// TIA Portal V16 export
// export: Created 2022-11-17T15:49:45.9581143Z, ExportSetting WithDefaults, DisplayName Totally Integrated Automation Portal, DisplayVersion V16 Update 6, DisplayName TIA Portal Version Control Interface, DisplayVersion V16 Update 2, DisplayName TIA Portal Openness, DisplayVersion V16 Update 6, DisplayName SINAMICS Startdrive Advanced, DisplayVersion V16 Update 5, DisplayName SINAMICS Startdrive G130, G150, S120, S150, SINAMICS MV, S210, DisplayVersion V16 Update 5, DisplayName SINAMICS Startdrive G110M, G120, G120C, G120D, G120P, G115D, DisplayVersion V16 Update 5, DisplayName STEP 7 Professional, DisplayVersion V16 Update 6, DisplayName STEP 7 Safety, DisplayVersion V16, DisplayName WinCC Advanced, DisplayVersion V16 Update 6
DATA_BLOCK "DB247_Program3"   // DB247
{ S7_Optimized_Access := 'FALSE' }
AUTHOR : Robopac
VERSION : 0.0
// stored: AutoNumber false, IsOnlyStoredInLoadMemory false, IsWriteProtectedInAS false
   VAR RETAIN
      Program3 { S7_SetPoint := 'True'} : "DatiProgramma";
   END_VAR
BEGIN
   Program3.Wrapping := TRUE;
   Program3.TopLenght := 500;
   Program3.TopRelease := 0;
   Program3.TopDown := 0;
   Program3.Top := 4;
   Program3.PressurePTime := 0;
   Program3.LifterTime := 0;
   Program3.RevOverContrast := 1;
   Program3.RopeEndCycle := 16#01;
   Program3.Spare4 := 16#01;
   Program3.RopeTime := 1500;
   Program3.RevOverClamp := 1;
   Program3.FilmForceFinalRev := 20;
   Program3.FilmPrestretchFinalRev := 100;
   Program3.ArmSpeed := 90;
   Program3.CarriageDown4Top := 500;
   Program3.TopDownTime := 1500;
   Program3.LapsUnderTop := 0;
   Program3.Spare6 := 0;
   Program3.Spare7 := 0;
   Program3.Spare8 := 0;
   Program3.Spare9 := 0;
   Program3.Spare10 := 0;
   Program3.Spare11 := 0;
   Program3.Spare12 := 0;
   Program3.Overlap0_1 := 0;
   Program3.Height1 := 120;
   Program3.Landmark1 := FALSE;
   Program3.Lifter1 := FALSE;
   Program3.SpareBit1H1 := FALSE;
   Program3.Airblower1 := TRUE;
   Program3.NextStep1 := TRUE;
   Program3.PressureP1 := TRUE;
   Program3.SpareByte2H1 := 16#00;
   Program3.Revolution1 := 1;
   Program3.RopeUnit1_1 := 16#01;
   Program3.RopeUnit1_2 := 16#01;
   Program3.FilmForce1 := 5;
   Program3.FilmPrestretch1 := 200;
   Program3.Spare3H1 := 0;
   Program3.Spare49 := 0;
   Program3.Spare50 := 0;
   Program3.Spare51 := 0;
   Program3.Spare52 := 0;
   Program3.Spare53 := 0;
   Program3.Overlap1_2 := 0;
   Program3.Height2 := 60;
   Program3.Landmark2 := FALSE;
   Program3.Lifter2 := FALSE;
   Program3.SpareBit1H2 := FALSE;
   Program3.Airblower2 := TRUE;
   Program3.NextStep2 := TRUE;
   Program3.PressureP2 := TRUE;
   Program3.SpareByte2H2 := 16#00;
   Program3.Revolution2 := 3;
   Program3.RopeUnit2_1 := 16#01;
   Program3.RopeUnit2_2 := 16#01;
   Program3.FilmForce2 := 10;
   Program3.FilmPrestretch2 := 200;
   Program3.Spare3H2 := 0;
   Program3.Spare54 := 0;
   Program3.Spare55 := 0;
   Program3.Spare56 := 0;
   Program3.Spare57 := 0;
   Program3.Spare58 := 0;
   Program3.Overlap2_3 := 100;
   Program3.Height3 := 120;
   Program3.Landmark3 := FALSE;
   Program3.Lifter3 := FALSE;
   Program3.SpareBit1H3 := FALSE;
   Program3.Airblower3 := TRUE;
   Program3.NextStep3 := TRUE;
   Program3.PressureP3 := TRUE;
   Program3.SpareByte2H3 := 16#00;
   Program3.Revolution3 := 2;
   Program3.RopeUnit3_1 := 16#01;
   Program3.RopeUnit3_2 := 16#01;
   Program3.FilmForce3 := 5;
   Program3.FilmPrestretch3 := 200;
   Program3.Spare3H3 := 0;
   Program3.Spare59 := 0;
   Program3.Spare60 := 0;
   Program3.Spare61 := 380;
   Program3.Spare62 := 2800;
   Program3.Spare63 := 0;
   Program3.Overlap3_4 := 200;
   Program3.Height4 := 120;
   Program3.Landmark4 := FALSE;
   Program3.Lifter4 := FALSE;
   Program3.SpareBit1H4 := FALSE;
   Program3.Airblower4 := TRUE;
   Program3.NextStep4 := TRUE;
   Program3.PressureP4 := TRUE;
   Program3.SpareByte2H4 := 16#00;
   Program3.Revolution4 := 1;
   Program3.RopeUnit4_1 := 16#01;
   Program3.RopeUnit4_2 := 16#01;
   Program3.FilmForce4 := 20;
   Program3.FilmPrestretch4 := 200;
   Program3.Spare3H4 := 0;
   Program3.Spare64 := 0;
   Program3.Spare65 := 0;
   Program3.Spare66 := 0;
   Program3.Spare67 := 0;
   Program3.Spare68 := 0;
   Program3.Overlap4_5 := 200;
   Program3.Height5 := -150;
   Program3.Landmark5 := TRUE;
   Program3.Lifter5 := FALSE;
   Program3.SpareBit1H5 := FALSE;
   Program3.Airblower5 := FALSE;
   Program3.NextStep5 := TRUE;
   Program3.PressureP5 := FALSE;
   Program3.SpareByte2H5 := 16#00;
   Program3.Revolution5 := 1;
   Program3.RopeUnit5_1 := 16#01;
   Program3.RopeUnit5_2 := 16#01;
   Program3.FilmForce5 := 20;
   Program3.FilmPrestretch5 := 200;
   Program3.Spare3H5 := 0;
   Program3.Spare69 := 0;
   Program3.Spare70 := 0;
   Program3.Spare71 := 0;
   Program3.Spare72 := 0;
   Program3.Spare73 := 0;
   Program3.Overlap5_6 := 100;
   Program3.Height6 := 0;
   Program3.Landmark6 := FALSE;
   Program3.Lifter6 := FALSE;
   Program3.SpareBit1H6 := FALSE;
   Program3.Airblower6 := FALSE;
   Program3.NextStep6 := FALSE;
   Program3.PressureP6 := FALSE;
   Program3.SpareByte2H6 := 16#00;
   Program3.Revolution6 := 1;
   Program3.RopeUnit6_1 := 16#01;
   Program3.RopeUnit6_2 := 16#01;
   Program3.FilmForce6 := 30;
   Program3.FilmPrestretch6 := 200;
   Program3.Spare3H6 := 0;
   Program3.Spare74 := 0;
   Program3.Spare75 := 0;
   Program3.Spare76 := 0;
   Program3.Spare77 := 0;
   Program3.Spare78 := 0;
   Program3.Overlap6_7 := 0;
   Program3.Height7 := 0;
   Program3.Landmark7 := FALSE;
   Program3.Lifter7 := FALSE;
   Program3.SpareBit1H7 := FALSE;
   Program3.Airblower7 := FALSE;
   Program3.NextStep7 := TRUE;
   Program3.PressureP7 := FALSE;
   Program3.SpareByte2H7 := 16#00;
   Program3.Revolution7 := 1;
   Program3.RopeUnit7_1 := 16#01;
   Program3.RopeUnit7_2 := 16#01;
   Program3.FilmForce7 := 0;
   Program3.FilmPrestretch7 := 100;
   Program3.Spare3H7 := 0;
   Program3.Spare79 := 0;
   Program3.Spare80 := 0;
   Program3.Spare81 := 0;
   Program3.Spare82 := 0;
   Program3.Spare83 := 0;
   Program3.Overlap7_8 := 0;
   Program3.Height8 := 0;
   Program3.Landmark8 := FALSE;
   Program3.Lifter8 := FALSE;
   Program3.SpareBit1H8 := FALSE;
   Program3.Airblower8 := FALSE;
   Program3.NextStep8 := TRUE;
   Program3.PressureP8 := FALSE;
   Program3.SpareByte2H8 := 16#00;
   Program3.Revolution8 := 1;
   Program3.RopeUnit8_1 := 16#01;
   Program3.RopeUnit8_2 := 16#01;
   Program3.FilmForce8 := 0;
   Program3.FilmPrestretch8 := 100;
   Program3.Spare3H8 := 0;
   Program3.Spare84 := 0;
   Program3.Spare85 := 0;
   Program3.Spare86 := 0;
   Program3.Spare87 := 0;
   Program3.Spare88 := 0;
   Program3.Overlap8_9 := 0;
   Program3.Height9 := 0;
   Program3.Landmark9 := FALSE;
   Program3.Lifter9 := FALSE;
   Program3.SpareBit1H9 := FALSE;
   Program3.Airblower9 := FALSE;
   Program3.NextStep9 := TRUE;
   Program3.PressureP9 := FALSE;
   Program3.SpareByte2H9 := 16#00;
   Program3.Revolution9 := 1;
   Program3.RopeUnit9_1 := 16#01;
   Program3.RopeUnit9_2 := 16#01;
   Program3.FilmForce9 := 0;
   Program3.FilmPrestretch9 := 100;
   Program3.Spare3H9 := 0;
   Program3.Spare89 := 0;
   Program3.Spare90 := 0;
   Program3.Spare91 := 0;
   Program3.Spare92 := 0;
   Program3.Spare93 := 0;
   Program3.Overlap9_10 := 0;
   Program3.Height10 := 0;
   Program3.Landmark10 := FALSE;
   Program3.Lifter10 := FALSE;
   Program3.SpareBit1H10 := FALSE;
   Program3.Airblower10 := FALSE;
   Program3.NextStep10 := FALSE;
   Program3.PressureP10 := FALSE;
   Program3.SpareByte2H10 := 16#00;
   Program3.Revolution10 := 1;
   Program3.RopeUnit10_1 := 16#01;
   Program3.RopeUnit10_2 := 16#01;
   Program3.FilmForce10 := 0;
   Program3.FilmPrestretch10 := 100;
   Program3.Spare3H10 := 0;
   Program3.Spare94 := 0;
   Program3.Spare95 := 0;
   Program3.Spare96 := 0;
   Program3.Spare97 := 0;
   Program3.Spare98 := 0;
   Program3.Overlap10_11 := 0;
   Program3.Height11 := 0;
   Program3.Landmark11 := FALSE;
   Program3.Lifter11 := FALSE;
   Program3.SpareBit1H11 := FALSE;
   Program3.Airblower11 := FALSE;
   Program3.NextStep11 := TRUE;
   Program3.PressureP11 := FALSE;
   Program3.SpareByte2H11 := 16#00;
   Program3.Revolution11 := 1;
   Program3.RopeUnit11_1 := 16#01;
   Program3.RopeUnit11_2 := 16#01;
   Program3.FilmForce11 := 0;
   Program3.FilmPrestretch11 := 100;
   Program3.Spare3H11 := 0;
   Program3.Spare99 := 0;
   Program3.Spare100 := 0;
   Program3.Spare101 := 0;
   Program3.Spare102 := 0;
   Program3.Spare103 := 0;
   Program3.Overlap11_12 := 0;
   Program3.Height12 := 0;
   Program3.Landmark12 := FALSE;
   Program3.Lifter12 := FALSE;
   Program3.SpareBit1H12 := FALSE;
   Program3.Airblower12 := FALSE;
   Program3.NextStep12 := FALSE;
   Program3.PressureP12 := FALSE;
   Program3.SpareByte2H12 := 16#00;
   Program3.Revolution12 := 1;
   Program3.RopeUnit12_1 := 16#01;
   Program3.RopeUnit12_2 := 16#01;
   Program3.FilmForce12 := 0;
   Program3.FilmPrestretch12 := 100;
   Program3.Spare3H12 := 0;
   Program3.Spare104 := 0;
   Program3.Spare105 := 0;
   Program3.Spare106 := 0;
   Program3.Spare107 := 0;
   Program3.Spare108 := 0;
END_DATA_BLOCK
